_CFC_ (* Continuous Function Chart, elements in execution order *)
#0 OR(SCHU_P2_2_UE1_T_RESET, SCHU_P2_2_SB)
#1 SEL(UE1_T_FILTER_ON, T#0ms, T#2s)
#2 fb_UE2_T:ISTOK_ANALOGVH(enable: TRUE, rawValue: SCHU_P2_2_UE1_AI1, reset: #0, enableLimitCtrl: enbleLimit, ctrlVoltage: NOT UE1_T_CVOLT, changeValueWithoutPower: TRUE, highRange: UE_T_HIGHRANGE, lowRange: UE_T_LOWRANGE, highLimit: SCHU_P2_2_UE_T_HIGHLIMIT, lowLimit: SCHU_P2_2_UE_T_LOWLIMIT, filterTime: #1, offset: ofset, delayEnable: TE_DELAY)
#3 SCHU_P2_2_UE1_T_VN <= #2.presentValue
#4 SCHU_P2_2_UE1_T_DOST <= #2.reliability
#5 SUB(SCHU_P2_2_UE1_T_UST, 0.6)
#6 fb_UE2_m_UST:ISTOK_LT(dost: #2.reliability, x: #2.presentValue, ust: #5, shkal: -, gist: 0.5)
#7 SCHU_P2_2_UE1_TE_M_UST <= #6.Xm
#8 SCHU_P2_2_UE1_TE_NM_UST <= #6.XmN
#9 ADD(SCHU_P2_2_UE1_T_UST, 0.6)
#10 fb_UE2_b_UST:ISTOK_GT(dost: #2.reliability, x: #2.presentValue, ust: #9, shkal: -, gist: 0.5)
#11 SCHU_P2_2_UE1_TE_B_UST <= #10.Xb
#12 SCHU_P2_2_UE1_TE_NB_UST <= #10.XbN
_END_CFC_
(* the same logic as Structured Text *)
fb_UE2_T(enable := TRUE, rawValue := SCHU_P2_2_UE1_AI1, reset := SCHU_P2_2_UE1_T_RESET OR SCHU_P2_2_SB, enableLimitCtrl := enbleLimit, ctrlVoltage := NOT UE1_T_CVOLT, changeValueWithoutPower := TRUE, highRange := UE_T_HIGHRANGE, lowRange := UE_T_LOWRANGE, highLimit := SCHU_P2_2_UE_T_HIGHLIMIT, lowLimit := SCHU_P2_2_UE_T_LOWLIMIT, filterTime := SEL(UE1_T_FILTER_ON, T#0ms, T#2s), offset := ofset, delayEnable := TE_DELAY);
SCHU_P2_2_UE1_T_VN := fb_UE2_T.presentValue;
SCHU_P2_2_UE1_T_DOST := fb_UE2_T.reliability;
fb_UE2_m_UST(dost := fb_UE2_T.reliability, x := fb_UE2_T.presentValue, ust := SCHU_P2_2_UE1_T_UST - 0.6, gist := 0.5);
SCHU_P2_2_UE1_TE_M_UST := fb_UE2_m_UST.Xm;
SCHU_P2_2_UE1_TE_NM_UST := fb_UE2_m_UST.XmN;
fb_UE2_b_UST(dost := fb_UE2_T.reliability, x := fb_UE2_T.presentValue, ust := SCHU_P2_2_UE1_T_UST + 0.6, gist := 0.5);
SCHU_P2_2_UE1_TE_B_UST := fb_UE2_b_UST.Xb;
SCHU_P2_2_UE1_TE_NB_UST := fb_UE2_b_UST.XbN;
END_PROGRAM

(* POU TZBiS/S/ALL_S, CFC *)
PROGRAM ALL_S
VAR
END_VAR
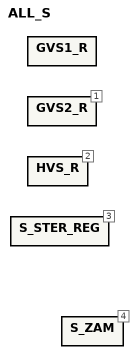
_CFC_ (* Continuous Function Chart, elements in execution order *)
#0 GVS1_R()
#1 GVS2_R()
#2 HVS_R()
#3 S_STER_REG()
#4 S_ZAM()
_END_CFC_
(* the same logic as Structured Text *)
GVS1_R();
GVS2_R();
HVS_R();
S_STER_REG();
S_ZAM();
END_PROGRAM

(* POU TZBiS/S/GVS1_R, CFC *)
PROGRAM GVS1_R
VAR
	rs_gvs1: RS;
	GVS1_RUN: BOOL;
END_VAR
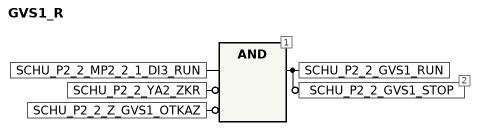
_CFC_ (* Continuous Function Chart, elements in execution order *)
#0 SCHU_P2_2_GVS1_RUN <= #1
#1 AND(SCHU_P2_2_MP2_2_1_DI3_RUN, NOT SCHU_P2_2_YA2_ZKR, NOT SCHU_P2_2_Z_GVS1_OTKAZ)
#2 SCHU_P2_2_GVS1_STOP <= NOT #1
_END_CFC_
END_PROGRAM

(* POU TZBiS/S/GVS2_R, CFC *)
PROGRAM GVS2_R
VAR
END_VAR
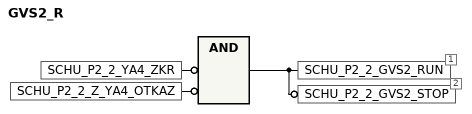
_CFC_ (* Continuous Function Chart, elements in execution order *)
#0 AND(NOT SCHU_P2_2_YA4_ZKR, NOT SCHU_P2_2_Z_YA4_OTKAZ)
#1 SCHU_P2_2_GVS2_RUN <= #0
#2 SCHU_P2_2_GVS2_STOP <= NOT #0
_END_CFC_
END_PROGRAM

(* POU TZBiS/S/HVS_R, CFC *)
PROGRAM HVS_R
VAR
END_VAR
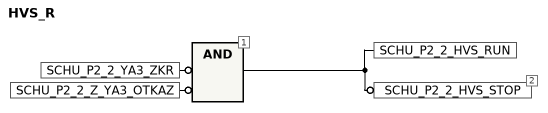
_CFC_ (* Continuous Function Chart, elements in execution order *)
#0 SCHU_P2_2_HVS_RUN <= #1
#1 AND(NOT SCHU_P2_2_YA3_ZKR, NOT SCHU_P2_2_Z_YA3_OTKAZ)
#2 SCHU_P2_2_HVS_STOP <= NOT #1
_END_CFC_
END_PROGRAM

(* POU TZBiS/S/S_STER_REG, CFC *)
PROGRAM S_STER_REG
VAR
	ZAD_S_Ster_Reg: TON;
END_VAR
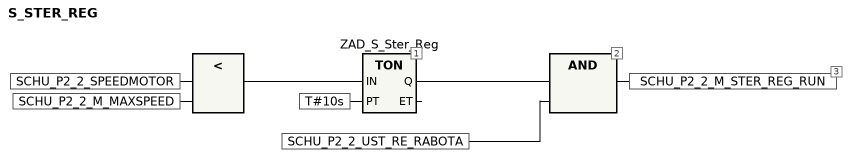
_CFC_ (* Continuous Function Chart, elements in execution order *)
#0 <(SCHU_P2_2_SPEEDMOTOR, SCHU_P2_2_M_MAXSPEED)
#1 ZAD_S_Ster_Reg:TON(IN: #0, PT: T#10s)
#2 AND(#1.Q, SCHU_P2_2_UST_RE_RABOTA)
#3 SCHU_P2_2_M_STER_REG_RUN <= #2
_END_CFC_
END_PROGRAM

(* POU TZBiS/S/S_ZAM, CFC *)
PROGRAM S_ZAM
VAR
	SR_ZAM: SR;
END_VAR
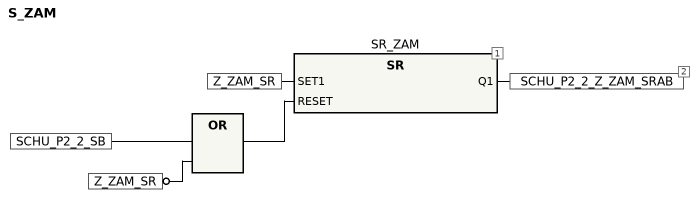
_CFC_ (* Continuous Function Chart, elements in execution order *)
#0 OR(SCHU_P2_2_SB, NOT Z_ZAM_SR)
#1 SR_ZAM:SR(SET1: Z_ZAM_SR, RESET: #0)
#2 SCHU_P2_2_Z_ZAM_SRAB <= #1.Q1
_END_CFC_
(* the same logic as Structured Text *)
SR_ZAM(SET1 := Z_ZAM_SR, RESET := SCHU_P2_2_SB OR NOT Z_ZAM_SR);
SCHU_P2_2_Z_ZAM_SRAB := SR_ZAM.Q1;
END_PROGRAM

(* POU TZBiS/TZB/ALL_TZB, CFC *)
PROGRAM ALL_TZB
VAR
END_VAR
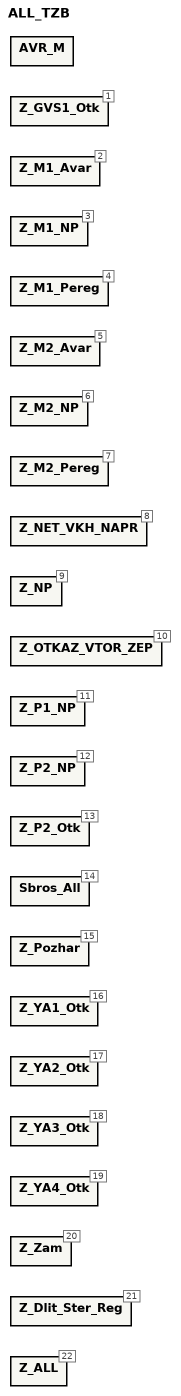
_CFC_ (* Continuous Function Chart, elements in execution order *)
#0 AVR_M()
#1 Z_GVS1_Otk()
#2 Z_M1_Avar()
#3 Z_M1_NP()
#4 Z_M1_Pereg()
#5 Z_M2_Avar()
#6 Z_M2_NP()
#7 Z_M2_Pereg()
#8 Z_NET_VKH_NAPR()
#9 Z_NP()
#10 Z_OTKAZ_VTOR_ZEP()
#11 Z_P1_NP()
#12 Z_P2_NP()
#13 Z_P2_Otk()
#14 Sbros_All()
#15 Z_Pozhar()
#16 Z_YA1_Otk()
#17 Z_YA2_Otk()
#18 Z_YA3_Otk()
#19 Z_YA4_Otk()
#20 Z_Zam()
#21 Z_Dlit_Ster_Reg()
#22 Z_ALL()
_END_CFC_
(* the same logic as Structured Text *)
AVR_M();
Z_GVS1_Otk();
Z_M1_Avar();
Z_M1_NP();
Z_M1_Pereg();
Z_M2_Avar();
Z_M2_NP();
Z_M2_Pereg();
Z_NET_VKH_NAPR();
Z_NP();
Z_OTKAZ_VTOR_ZEP();
Z_P1_NP();
Z_P2_NP();
Z_P2_Otk();
Sbros_All();
Z_Pozhar();
Z_YA1_Otk();
Z_YA2_Otk();
Z_YA3_Otk();
Z_YA4_Otk();
Z_Zam();
Z_Dlit_Ster_Reg();
Z_ALL();
END_PROGRAM

(* POU TZBiS/TZB/AVR_M, CFC *)
PROGRAM AVR_M
VAR
	fb_HVACRC: FB_HVACRedundancyCtrl;
	RS_Pusk: RS;
	RT_Pusk: R_TRIG;


	rHours: ARRAY[1..8] OF REAL;
	uiCount: ARRAY[1..8] OF UINT;

	delayFBC: TIME := T#1s;
	overlap1Actuator: TIME := T#0s;
	maxOnLevel: UINT := 12;

	dtSystemTime: DT;
	fb_HVAC_GST: FB_HVACGetSystemTime;
	error: BOOL;
	RS_avr_kom: RS;
	RT_T: R_TRIG;
	TON_VKL: TON;
	TON_PUSK: TON;
END_VAR
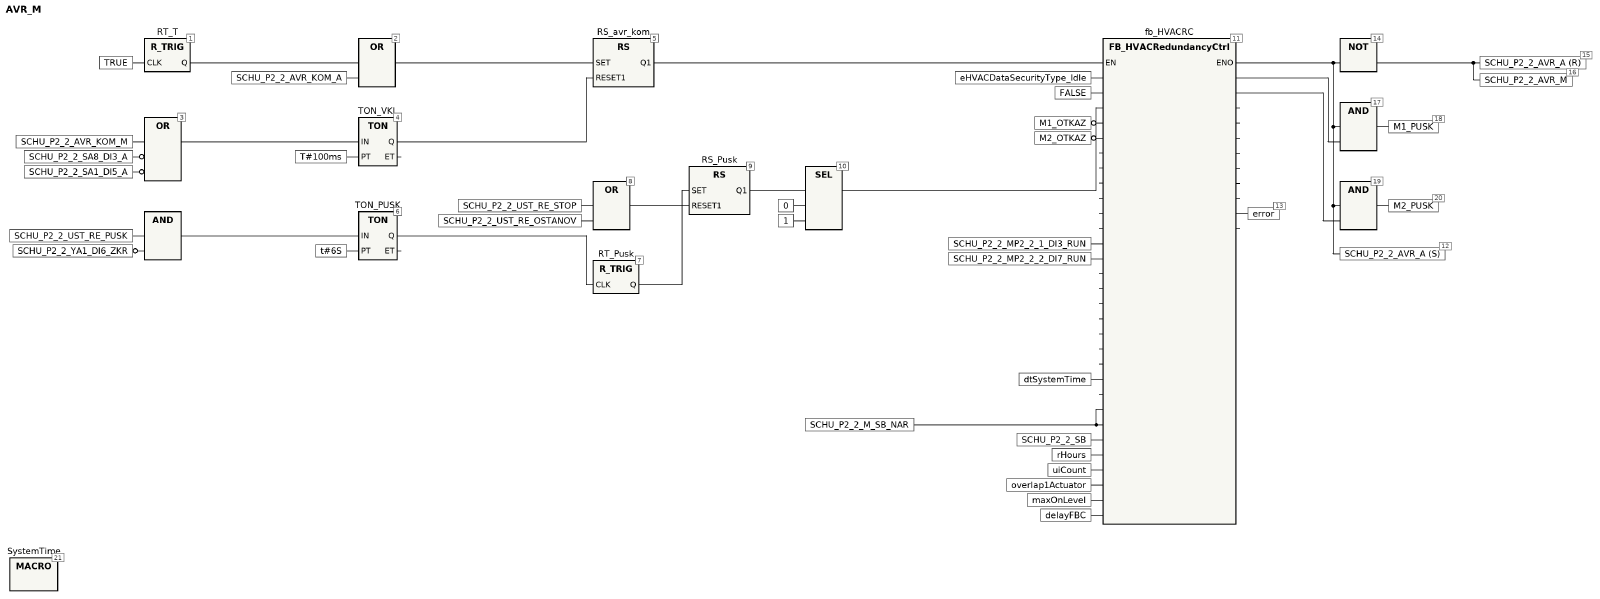
